FUNCTION_BLOCK TaurusLed IMPLEMENTS I_TaurusLed
VAR
	_text AT%M* 		: T_MaxString;

	forwardButton		: I_Button;
	motorTermFuse		: I_TermFuse;
	statusScadaLabel	: I_Label;
	
END_VAR

// ustaw stan zmiennej LED Taurusa w TANGO SCADA


statusScadaLabel.Text := 'ON';	

IF motorTermFuse.IsActive THEN
		_text := 'ON';
		statusScadaLabel.Text := 'ON';	
	IF forwardButton.IsPressed THEN
		_text := 'RUNNING';
		statusScadaLabel.Text := 'RUNNING';
	END_IF
ELSE
		_text := 'OFF';
		statusScadaLabel.Text := 'OFF';
	IF forwardButton.IsPressed THEN
		_text := 'FAULT';
		statusScadaLabel.Text := 'FAULT';
	END_IF
END_IF

METHOD FB_init : BOOL
VAR_INPUT
	bInitRetains 		: BOOL; // if TRUE, the retain variables are initialized (warm start / cold start)
	bInCopyCode 		: BOOL;  // if TRUE, the instance afterwards gets moved into the copy code (online change)
	forwardButton		: I_Button;
	motorTermFuse		: I_TermFuse;
	statusScadaLabel	: I_Label;
END_VAR
THIS^.forwardButton			:= forwardButton;
THIS^.motorTermFuse			:= motorTermFuse;
THIS^.statusScadaLabel      := statusScadaLabel;
END_METHOD

PROPERTY Text : STRING
GET
Text := _text;
END_GET
SET
_text := Text;
END_SET
END_PROPERTY

END_FUNCTION_BLOCK

(* stored: Version 1.1.0.1, ProductVersion 3.1.4024.12
   POU TaurusLed: Id {f6f49f3d-8a72-4f7a-b651-4716ce5ac1db}, SpecialFunc None
   Method FB_init: Id {73c97024-5816-4e10-b55f-f67168980634}
   Property Text: Id {1aa88967-6225-4ffd-82b4-3b009d2bfb86}
   Get Get: Id {60d7d138-8c96-4745-b0e3-e36305ce1073}
   Set Set: Id {4611a705-c695-4abd-9093-7cf7b6a5ad8d} *)
